FUNCTION_BLOCK ElevatoriaEsgotoBruto (* Composite Function Block Type *)
  (* Standard: 61499-2 *)
  (* Version 0.0, 24/02/2026, template *)
  PACKAGE Hidryco.HidrycoLib;
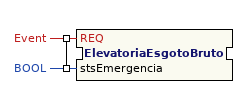
  EVENT_INPUT
    REQ WITH stsEmergencia;
  END_EVENT
  VAR_INPUT
    stsEmergencia : BOOL;
  END_VAR
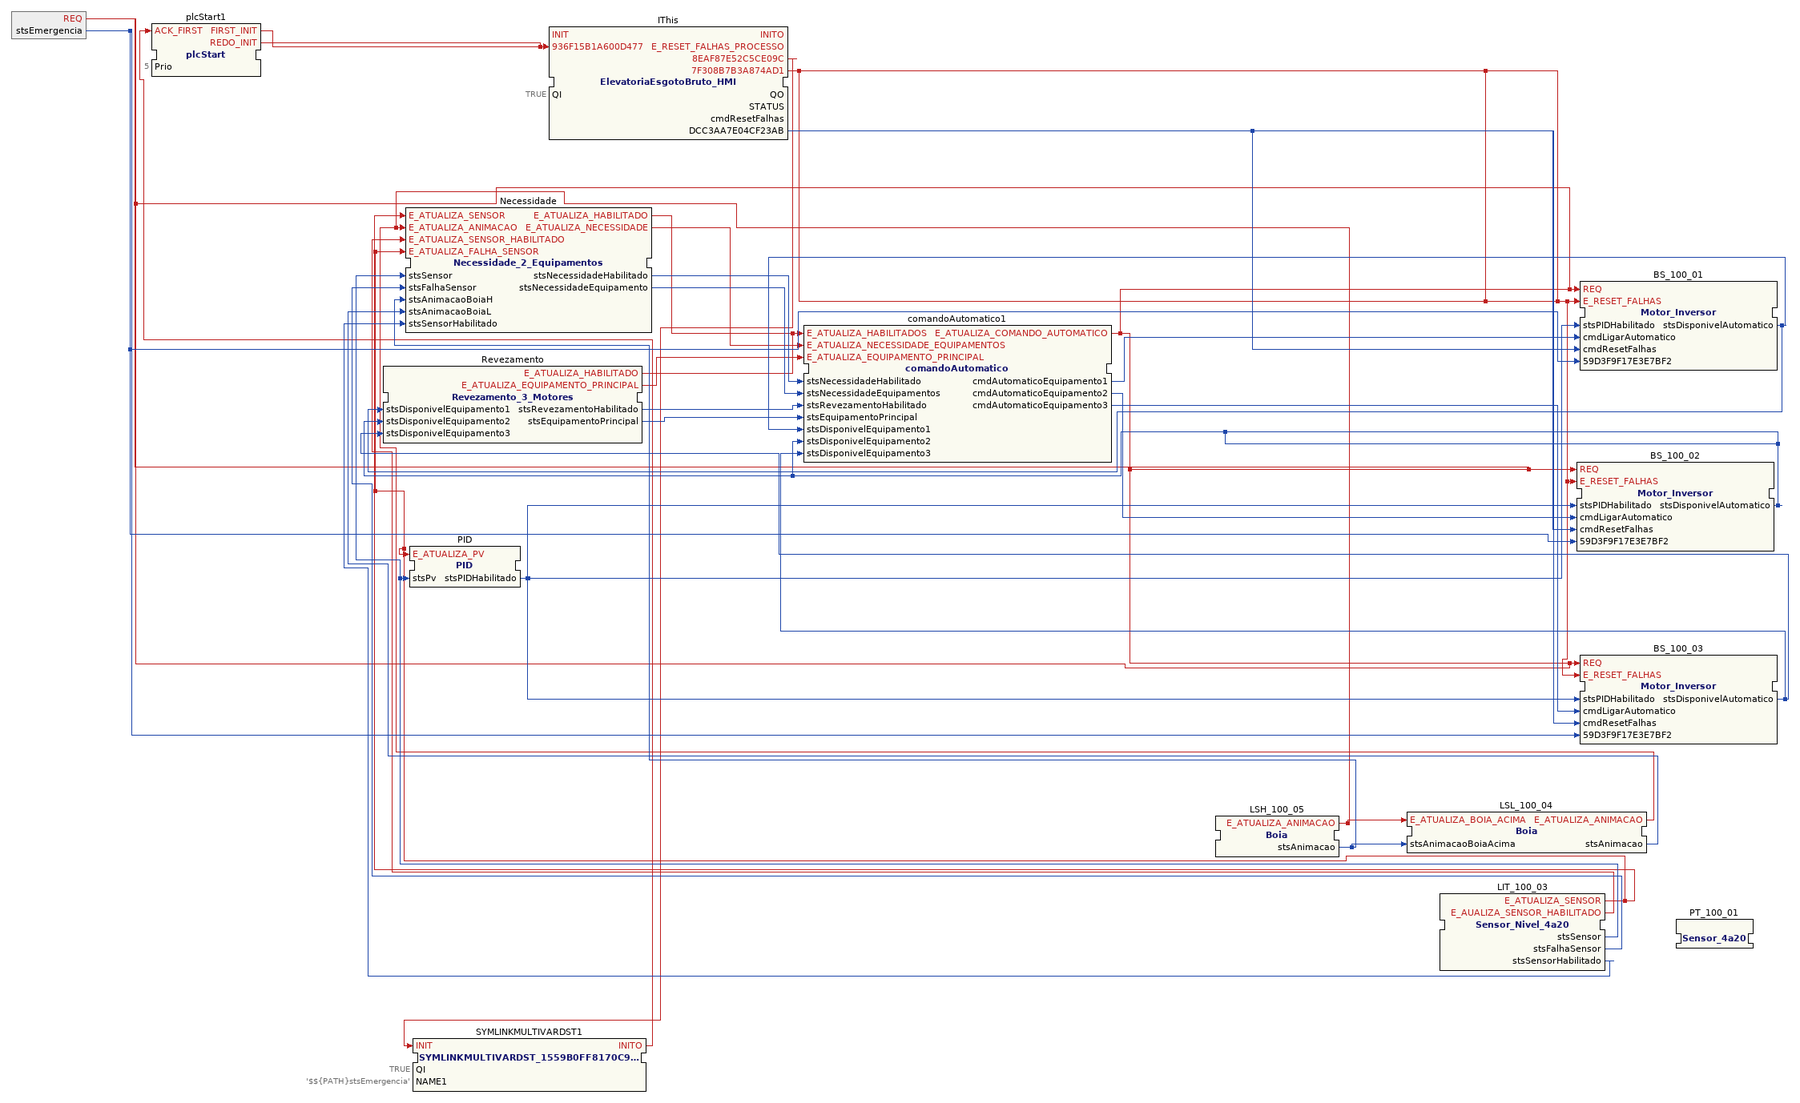
  (* 0 - INITIALIZATION *)
  (* 1 - FUNCTIONAL INPUT INTERFACE *)
  (* 6 - OT-IT INTERFACE *)
  (* 2 - FUNCTIONAL OUTPUT INTERFACE *)
  (* 3 - FIELD INTERFACE *)
  (* 4 - CHILDREN *)
  (* 5 - LOGICS *)
  (* 5.B - OPERATION MODE MANAGEMENT *)
  (* 5.C - INTERLOCKS MANAGEMENT *)
  (* 5.A - FUNCTIONAL BEHAVIORS *)
  FBS
    LSH_100_05 : Boia; {SET_ATTRIBUTE(Configuration.Component.HideUnusedPorts, )}
    LSL_100_04 : Boia;
    BS_100_01 : Motor_Inversor;
    BS_100_02 : Motor_Inversor;
    BS_100_03 : Motor_Inversor;
    plcStart1 : plcStart(Prio := 5);
    SYMLINKMULTIVARDST1 : SYMLINKMULTIVARDST_1559B0FF8170C9BA0(QI := TRUE, NAME1 := '$${PATH}stsEmergencia'); {SET_ATTRIBUTE(Configuration.GenericFBType.InterfaceParams, Runtime.System#I:=1;VALUE${I$}:BOOL)}
    PID : PID;
    Revezamento : Revezamento_3_Motores;
    Necessidade : Necessidade_2_Equipamentos;
    comandoAutomatico1 : comandoAutomatico;
    IThis : ElevatoriaEsgotoBruto_HMI(QI := TRUE);
    PT_100_01 : Sensor_4a20;
    LIT_100_03 : Sensor_Nivel_4a20;
  END_FBS
  EVENT_CONNECTIONS
    LSH_100_05.E_ATUALIZA_ANIMACAO TO LSL_100_04.E_ATUALIZA_BOIA_ACIMA;
    LIT_100_03.E_ATUALIZA_SENSOR TO PID.E_ATUALIZA_PV;
    Necessidade.E_ATUALIZA_HABILITADO TO comandoAutomatico1.E_ATUALIZA_HABILITADOS;
    Revezamento.E_ATUALIZA_HABILITADO TO comandoAutomatico1.E_ATUALIZA_HABILITADOS;
    Necessidade.E_ATUALIZA_NECESSIDADE TO comandoAutomatico1.E_ATUALIZA_NECESSIDADE_EQUIPAMENTOS;
    LIT_100_03.E_ATUALIZA_SENSOR TO Necessidade.E_ATUALIZA_SENSOR;
    LSH_100_05.E_ATUALIZA_ANIMACAO TO Necessidade.E_ATUALIZA_ANIMACAO;
    LSL_100_04.E_ATUALIZA_ANIMACAO TO Necessidade.E_ATUALIZA_ANIMACAO;
    Revezamento.E_ATUALIZA_EQUIPAMENTO_PRINCIPAL TO comandoAutomatico1.E_ATUALIZA_EQUIPAMENTO_PRINCIPAL;
    comandoAutomatico1.E_ATUALIZA_COMANDO_AUTOMATICO TO BS_100_01.REQ;
    comandoAutomatico1.E_ATUALIZA_COMANDO_AUTOMATICO TO BS_100_02.REQ;
    comandoAutomatico1.E_ATUALIZA_COMANDO_AUTOMATICO TO BS_100_03.REQ;
    plcStart1.FIRST_INIT TO IThis.936F15B1A600D477;
    plcStart1.REDO_INIT TO IThis.936F15B1A600D477;
    SYMLINKMULTIVARDST1.INITO TO plcStart1.ACK_FIRST;
    IThis.8EAF87E52C5CE09C TO SYMLINKMULTIVARDST1.INIT;
    IThis.7F308B7B3A874AD1 TO BS_100_01.E_RESET_FALHAS;
    IThis.7F308B7B3A874AD1 TO BS_100_02.E_RESET_FALHAS;
    IThis.7F308B7B3A874AD1 TO BS_100_03.E_RESET_FALHAS;
    LIT_100_03.E_AUALIZA_SENSOR_HABILITADO TO Necessidade.E_ATUALIZA_SENSOR_HABILITADO;
    REQ TO BS_100_01.REQ;
    REQ TO BS_100_02.REQ;
    REQ TO BS_100_03.REQ;
    LIT_100_03.E_ATUALIZA_SENSOR TO Necessidade.E_ATUALIZA_FALHA_SENSOR;
  END_CONNECTIONS
  DATA_CONNECTIONS
    LIT_100_03.stsSensor TO PID.stsPv;
    PID.stsPIDHabilitado TO BS_100_01.stsPIDHabilitado;
    PID.stsPIDHabilitado TO BS_100_02.stsPIDHabilitado;
    PID.stsPIDHabilitado TO BS_100_03.stsPIDHabilitado;
    BS_100_01.stsDisponivelAutomatico TO Revezamento.stsDisponivelEquipamento1;
    BS_100_02.stsDisponivelAutomatico TO Revezamento.stsDisponivelEquipamento2;
    BS_100_03.stsDisponivelAutomatico TO Revezamento.stsDisponivelEquipamento3;
    LSH_100_05.stsAnimacao TO LSL_100_04.stsAnimacaoBoiaAcima;
    Necessidade.stsNecessidadeHabilitado TO comandoAutomatico1.stsNecessidadeHabilitado;
    Necessidade.stsNecessidadeEquipamento TO comandoAutomatico1.stsNecessidadeEquipamentos;
    Revezamento.stsRevezamentoHabilitado TO comandoAutomatico1.stsRevezamentoHabilitado;
    Revezamento.stsEquipamentoPrincipal TO comandoAutomatico1.stsEquipamentoPrincipal;
    BS_100_01.stsDisponivelAutomatico TO comandoAutomatico1.stsDisponivelEquipamento1;
    BS_100_02.stsDisponivelAutomatico TO comandoAutomatico1.stsDisponivelEquipamento2;
    BS_100_03.stsDisponivelAutomatico TO comandoAutomatico1.stsDisponivelEquipamento3;
    comandoAutomatico1.cmdAutomaticoEquipamento1 TO BS_100_01.cmdLigarAutomatico;
    comandoAutomatico1.cmdAutomaticoEquipamento2 TO BS_100_02.cmdLigarAutomatico;
    comandoAutomatico1.cmdAutomaticoEquipamento3 TO BS_100_03.cmdLigarAutomatico;
    LIT_100_03.stsSensor TO Necessidade.stsSensor;
    LIT_100_03.stsFalhaSensor TO Necessidade.stsFalhaSensor;
    LSH_100_05.stsAnimacao TO Necessidade.stsAnimacaoBoiaH;
    LSL_100_04.stsAnimacao TO Necessidade.stsAnimacaoBoiaL;
    IThis.DCC3AA7E04CF23AB TO BS_100_01.cmdResetFalhas;
    IThis.DCC3AA7E04CF23AB TO BS_100_02.cmdResetFalhas;
    IThis.DCC3AA7E04CF23AB TO BS_100_03.cmdResetFalhas;
    LIT_100_03.stsSensorHabilitado TO Necessidade.stsSensorHabilitado;
    stsEmergencia TO BS_100_01.59D3F9F17E3E7BF2;
    stsEmergencia TO BS_100_02.59D3F9F17E3E7BF2;
    stsEmergencia TO BS_100_03.59D3F9F17E3E7BF2;
  END_CONNECTIONS
END_FUNCTION_BLOCK
